FUNCTION_BLOCK Process EXTENDS Station IMPLEMENTS IProcess
VAR_INPUT
END_VAR
VAR_OUTPUT
END_VAR
VAR
	_isProcess : BOOL;
	_startPos : MC_LREAL;
	_endPos : MC_LREAL;
	_processVelo : MC_LREAL;
END_VAR

IF _isProcess THEN
	;
ELSE
	SUPER^();
END_IF

PROPERTY EndPosition : MC_LREAL
GET
EndPosition := _endPos;
END_GET
SET
_endPos := EndPosition;
END_SET
END_PROPERTY

{warning 'add property implementation'}
PROPERTY IsProcess : BOOL
GET
IsProcess := _isProcess;
END_GET
SET
_isProcess := IsProcess;
END_SET
END_PROPERTY

PROPERTY ProcessVelocity : MC_LREAL
GET
ProcessVelocity := _processVelo;
END_GET
SET
_processVelo := ProcessVelocity;
END_SET
END_PROPERTY

PROPERTY StartPosition : MC_LREAL
GET
StartPosition := _startPos;
END_GET
SET
_startPos := StartPosition;
END_SET
END_PROPERTY

END_FUNCTION_BLOCK

(* stored: Version 1.1.0.1, ProductVersion 3.1.4024.9
   POU Process: Id {6ff66696-ca88-4741-8ceb-6eabe3db4358}, SpecialFunc None
   Property EndPosition: Id {34687522-c87a-450b-8fec-5eba5de4d8e4}
   Get Get: Id {3d4b6083-f8e7-4e42-b785-f926e0e4624b}
   Set Set: Id {71ea4e89-2d7b-4ea4-bc43-277fa217fe85}
   Property IsProcess: Id {64c45dba-15e3-4d6e-bd80-f5540438ff58}
   Get Get: Id {ca66241c-5fea-4834-a0ef-193c14c3abcd}
   Set Set: Id {819910c6-3d14-4eb8-b190-1393e913f8da}
   Property ProcessVelocity: Id {be841438-829c-4b26-a447-921f37e8e334}
   Get Get: Id {3671f696-a3b4-4b45-9710-4a8de1678aae}
   Set Set: Id {204837d6-670b-4068-bdeb-608614eb83d9}
   Property StartPosition: Id {e538eeca-f7a3-4ed3-8499-b2ced4d78d04}
   Get Get: Id {a9e26d3c-c88b-4ccf-a30b-4912df977429}
   Set Set: Id {09a2c929-42e1-432d-a774-db779c301003} *)
